PROGRAM SlowPRG_1
VAR
	bolPlcStartupDone: BOOL := FALSE;
	bolHostInitDone: BOOL := FALSE;
	bolInitDone: BOOL := FALSE;
	uinTaskNbr : UINT := 3; // SlowTask is Task Nr 3
	jj:INT;
	bolCtrlRst: BOOL;		// Global alarm reset for ICL
	bolSimulateAll: BOOL; // Switches all controllers in ICL to simulation with pos. edge
	bolSimulationActive: BOOL;

		
	FUB_ICL_TEST : 	FB_ICL();
	stSequence : T_Sequence;
	pFB_Test: POINTER TO FB_STB;
	pFB_Test1: POINTER TO FB_MER;
	pFB_Test2: POINTER TO IBuffer;
	//pFB_Test2: POINTER TO TestIBuffer;
	pFB_Test3: POINTER TO FB_IBuffer;
	IChildTypeIBuffer: IBuffer;
	
	fbAlm_Man: FB_Alm_Man; // alarm manager

END_VAR

(*__________________________________________________________________________________________________
¦	
¦	Vistaprint Schweiz GmbH
¦	CH - 8401 Winterthur
¦
¦	www.vistaprint.ch - info@vistaprint.ch
¦___________________________________________________________________________________________________

Function desription:
call of all controller (FUB) for the slow task class.


History:
Version		Date			Author		Comment
---------------------------------------------------------------------------------------------------
0.00.1		06.09.2013		AVME/KVO	Start history
0.00.2		21.11.2013		AVME/MRU	Use BaseHts as Lib, StartUp Order
0.00.3		29.11.2013		AVME/MRU	Some Bugs fixed in IoInBridge
0.00.4		02.12.2013		AVME/MRU	Remove CurrentItemCounter and some Bugs fixed

___________________________________________________________________________________________________*)

// -----------------------------------------------------------------------------------------------
// Initialize the PLC Parameter and check the PLC health
// -----------------------------------------------------------------------------------------------
IF ((NOT bolPlcStartupDone) AND (g_uinStartProzess>=(uinTaskNbr-1))) THEN
	bolPlcStartupDone := TRUE;	
		
	// init	
	FUB_ICL_TEST.iniAllCtrlArrays(ADR(g_a_pCtrlInst),ADR(g_a_pCtrlCIf),E_CtrlId.ICL_1); 

	// New run Group 2 starts here!
	FUB_ICL_TEST.AddRunGrpTime(2000); // Wait 2sec before change to next group
	// New stop Group 2 starts here!
	FUB_ICL_TEST.AddStopGrpTime(6000); // Wait 6sec before change to next group
	// New run Group 3 starts here!
	FUB_ICL_TEST.AddRunGrpTime(8000); // Wait 8sec before change to next group
	// New stop Group 3 starts here!
	FUB_ICL_TEST.AddStopGrpTime(6000); // Wait 6sec before change to next group
	// New run Group 4 starts here!
	FUB_ICL_TEST.AddRunGrpTime(8000); // Wait 8sec before change to next group
	// New stop Group 4 starts here!
	FUB_ICL_TEST.AddStopGrpTime(6000); // Wait 6sec before change to next group
		
	// Define sequence parameter
	stSequence.pChild:= g_a_pCtrlInst[E_CtrlId.TLC_2];
	stSequence.uinGroupRun:= 1;
	stSequence.uinGroupStop:= 1;	
	stSequence.intCmdSeqRun:= cCMD_RUN;
	stSequence.intStatusSeqRun:= cSTA_RUN;
	stSequence.intCmdSeqStop:= cCMD_OFF;
	stSequence.intStatusSeqStop:= cSTA_OFF;
	// Add sequence group
	FUB_ICL_TEST.AddSeqChild(stSequence);
	
	// Define sequence parameter
	stSequence.pChild:= g_a_pCtrlInst[E_CtrlId.TLP_4];
	stSequence.uinGroupRun:= 2;
	stSequence.uinGroupStop:= 1;	
	stSequence.intCmdSeqRun:= cCMD_RUN;
	stSequence.intStatusSeqRun:= cSTA_RUN;
	stSequence.intCmdSeqStop:= cCMD_OFF;
	stSequence.intStatusSeqStop:= cSTA_OFF;
	// Add sequence group
	FUB_ICL_TEST.AddSeqChild(stSequence);

	// Define sequence parameter
	stSequence.pChild:= g_a_pCtrlInst[E_CtrlId.TLP_5];
	stSequence.uinGroupRun:= 3;
	stSequence.uinGroupStop:= 2;	
	stSequence.intCmdSeqRun:= cCMD_RUN;
	stSequence.intStatusSeqRun:= cSTA_RUN;
	stSequence.intCmdSeqStop:= cCMD_OFF;
	stSequence.intStatusSeqStop:= cSTA_OFF;
	// Add sequence group
	FUB_ICL_TEST.AddSeqChild(stSequence);
	
	// Define sequence parameter
	stSequence.pChild:= g_a_pCtrlInst[E_CtrlId.TLK_9];
	stSequence.uinGroupRun:= 4;
	stSequence.uinGroupStop:= 3;	
	stSequence.intCmdSeqRun:= cCMD_RUN;
	stSequence.intStatusSeqRun:= cSTA_RUN;
	stSequence.intCmdSeqStop:= cCMD_OFF;
	stSequence.intStatusSeqStop:= cSTA_OFF;
	// Add sequence group
	FUB_ICL_TEST.AddSeqChild(stSequence);

	// Add buffer elements
	FUB_ICL_TEST.AddIBufferChilds(g_a_pCtrlInst[E_CtrlId.SEP_2]); 
	FUB_ICL_TEST.AddIBufferChilds(g_a_pCtrlInst[E_CtrlId.DSB_2]); 
	FUB_ICL_TEST.AddIBufferChilds(g_a_pCtrlInst[E_CtrlId.SBI_5]); 
	FUB_ICL_TEST.AddIBufferChilds(g_a_pCtrlInst[E_CtrlId.DBO_5]); 
	FUB_ICL_TEST.AddIBufferChilds(g_a_pCtrlInst[E_CtrlId.SBI_3]); 
	FUB_ICL_TEST.AddIBufferChilds(g_a_pCtrlInst[E_CtrlId.BUF_10]); 
	FUB_ICL_TEST.AddIBufferChilds(g_a_pCtrlInst[E_CtrlId.SLB_8]); 

	g_uinStartProzess := g_uinStartProzess + 1;	// For StartUp order
	
END_IF
// -----------------------------------------------------------------------------------------------


// -----------------------------------------------------------------------------------------------
// The host system is downloading all parameter at startup. 
// bolPlcStartupDone will be set to true after the Host is done with the initialization
// -----------------------------------------------------------------------------------------------
IF (bolPlcStartupDone AND (NOT bolHostInitDone) AND (NOT bolInitDone)AND (g_uinStartProzess>=(uinTaskNbr-1)+10)) THEN

	// set all initialized controller FB the property of the alarm manager adress 
    Base_PLC.setAllCtrlAlarmFB(pCtrlInst := ADR(g_a_pCtrlInst[0]), pAlarmCtrl := ADR(fbAlm_Man), uinCtrlInstLength := INT_TO_UINT(E_CtrlId.E_CtrlIdMax));
    g_p_fbAlm_Man := ADR(fbAlm_Man); 

	g_uinStartProzess := g_uinStartProzess + 1;	// For StartUp order
	bolHostInitDone := TRUE;
END_IF
// -----------------------------------------------------------------------------------------------


// -----------------------------------------------------------------------------------------------
// Start PLC code initialization
// -----------------------------------------------------------------------------------------------
IF NOT bolInitDone AND bolPlcStartupDone AND bolHostInitDone AND (g_uinStartProzess>=(uinTaskNbr-1)+20) THEN
	g_uinStartProzess := g_uinStartProzess + 1;	// For StartUp order
	bolInitDone := TRUE;
END_IF
// -----------------------------------------------------------------------------------------------

// -----------------------------------------------------------------------------------------------
// Normal Run mode after all the initialization is done
// -----------------------------------------------------------------------------------------------
IF (bolInitDone AND bolPlcStartupDone AND bolHostInitDone AND (g_uinStartProzess>=(20+c_uinCntTaskClass))) THEN
	

	//****************************************************************************************************
	// SIMULATE all controller
	//****************************************************************************************************
	
	IF (bolSimulateAll = TRUE) AND (bolSimulationActive = FALSE) THEN
		// Enable simulation for all controller	
		FOR jj:=0 TO E_CtrlId.E_CtrlIdMax BY 1 DO
			IF (g_a_pCtrlCIf[jj]<>0) THEN // check if entry exist
				g_a_pCtrlCIf[jj]^.SwCfg.bolSimulation := TRUE;
			END_IF
		END_FOR	
		bolSimulationActive:= TRUE;
		// Trigger an alarm reset
		bolCtrlRst:= TRUE;
	END_IF
		
	IF (bolSimulateAll = FALSE) AND (bolSimulationActive = TRUE) THEN
		// Disable simulation for all controller	
		FOR jj:=0 TO E_CtrlId.E_CtrlIdMax BY 1 DO
			IF (g_a_pCtrlCIf[jj]<>0) THEN // check if entry exist
				g_a_pCtrlCIf[jj]^.SwCfg.bolSimulation := FALSE;
			END_IF
		END_FOR	
		bolSimulationActive:= FALSE;		
	END_IF

	//****************************************************************************************************
	// call alarm message handler
	//****************************************************************************************************
	fbAlm_Man(bolCtrlRst:= bolCtrlRst);
	IF (bolCtrlRst) THEN
		FOR jj:=0 TO E_CtrlId.E_CtrlIdMax BY 1 DO
			IF (g_a_pCtrlCIf[jj]<>0) THEN // check if entry exist
				g_a_pCtrlCIf[jj]^.Job.bolAlmReset := TRUE;
			END_IF
		END_FOR
		bolCtrlRst := FALSE;
	END_IF



	//FB_Test();
	FUB_ICL_TEST();

END_IF
// -----------------------------------------------------------------------------------------------

END_PROGRAM

(* stored: Version 1.1.0.1, ProductVersion 3.1.0.19
   POU SlowPRG_1: Id {1880a415-9f7f-4d4a-ad15-2dcfa97d058e} *)
